Staubli VAL3: readRect.pgx

public program readRect(num x_nCamID (dimensions=1), string x_sCellNumber (dimensions=1), trsf& x_trOrigin[] (dimensions=1), trsf& x_trSize[] (dimensions=1), bool& x_bError[] (dimensions=1))
  local bool l_bIsOk
  local string l_sColumn
  local string l_sMsgError
begin
  //-----------------------------------------------------------------------
  //Header begin
  //Description of program
  //  Read rectangle information from cells addressed by x_sCellNumber from
  //  camera' ID. Information must be stored in five consecutive cells
  //  in a row starting from x_sCellNumber : x, y, width, height and rz.
  //  - x, y and rz describe the position and rotation of the rectangle
  //  and are returned in x_trOrigin.
  //  - width (x) and height (y) describe the size of the rectangle and are
  //  returned in x_trSize.
  //
  //Input parameters
  //  num x_nCamID :
  //    role : camera's ID
  //  string x_sCellNumber :
  //    role : column of cell to read ("A1" or "B5" ...)
  //
  //Output parameters
  //  trsf x_trOrigin :
  //    role : position and rotation of the rectangle
  //  trsf x_trSize
  //    role : describe the size of the rectangle
  //  bool x_bError :
  //    role : returns true if an error occurred and false otherwise
  //
  //Examples
  //  call readRect(nCamID,"D5",l_trOrigine,l_trSize,l_bError)
  //
  //History
  //  Creation : 19-05-08 - f.Rob
  //Header end
  //----------------------------------------------------------------------

  x_bError=true
  // Read X coordinate from spreadsheet
  call readNumValue(x_nCamID,x_sCellNumber,x_trOrigin.x,x_bError)
  if !x_bError
    // Increment column number
    call incrementCol(x_sCellNumber,l_bIsOk)
    if l_bIsOk
      // Read Y coordinate from spreadsheet
      call readNumValue(x_nCamID,x_sCellNumber,x_trOrigin.y,x_bError)
      if !x_bError
        // Read width from spreadsheet
        call incrementCol(x_sCellNumber,l_bIsOk)
        if l_bIsOk
          call readNumValue(x_nCamID,x_sCellNumber,x_trSize.x,x_bError)
          if !x_bError
            // Read height from spreadsheet
            call incrementCol(x_sCellNumber,l_bIsOk)
            call readNumValue(x_nCamID,x_sCellNumber,x_trSize.y,x_bError)
            if !x_bError
              // Read RZ from spreadsheet
              call incrementCol(x_sCellNumber,l_bIsOk)
              if l_bIsOk
                call readNumValue(x_nCamID,x_sCellNumber,x_trOrigin.rz,x_bError)
              endIf
            endIf
          endIf
        endIf
      endIf
    endIf
  endIf
end
